{attribute 'pack_mode' := '1'}
TYPE IncomingMessage :
STRUCT
	id: MessageID;   (* Used to identify new messages. *)
	version: LINT;   (* Matches serialVersionUID of the equivalent Java class. *)
END_STRUCT
END_TYPE

(* stored: Version 1.1.0.1, ProductVersion 3.1.4022.12
   DUT IncomingMessage: Id {3726b91a-f9a9-45ea-9098-fc46e3b52a33} *)
